// Mitsubishi GX Works2 project: Project   PLC: Q00U

PROGRAM Conveyor
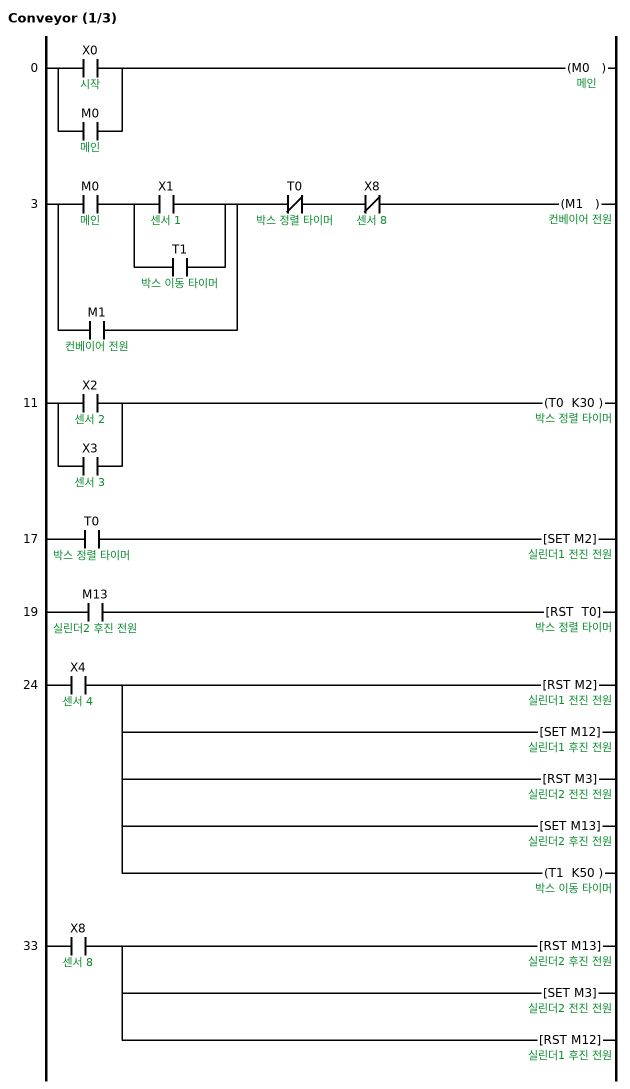
0     LD      X0  ; 시작
      OR      M0  ; 메인
      OUT     M0  ; 메인
3     LD      M0  ; 메인
      LD      X1  ; 센서 1
      OR      T1  ; 박스 이동 타이머
      ANB
      OR      M1  ; 컨베이어 전원
      ANI     T0  ; 박스 정렬 타이머
      ANI     X8  ; 센서 8
      OUT     M1  ; 컨베이어 전원
11    LD      X2  ; 센서 2
      OR      X3  ; 센서 3
      OUT     T0 K30  ; 박스 정렬 타이머
17    LD      T0  ; 박스 정렬 타이머
      SET     M2  ; 실린더1 전진 전원
19    LD      M13  ; 실린더2 후진 전원
      RST     T0  ; 박스 정렬 타이머
24    LD      X4  ; 센서 4
      RST     M2  ; 실린더1 전진 전원
      SET     M12  ; 실린더1 후진 전원
      RST     M3  ; 실린더2 전진 전원
      SET     M13  ; 실린더2 후진 전원
      OUT     T1 K50  ; 박스 이동 타이머
33    LD      X8  ; 센서 8
      RST     M13  ; 실린더2 후진 전원
      SET     M3  ; 실린더2 전진 전원
      RST     M12  ; 실린더1 후진 전원
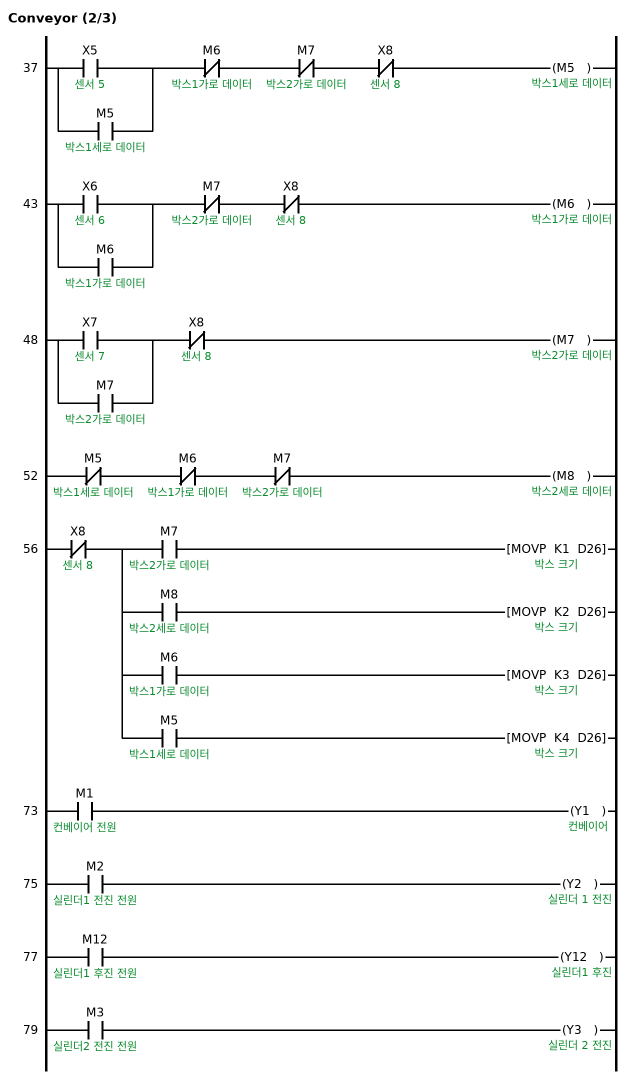
37    LD      X5  ; 센서 5
      OR      M5  ; 박스1세로 데이터
      ANI     M6  ; 박스1가로 데이터
      ANI     M7  ; 박스2가로 데이터
      ANI     X8  ; 센서 8
      OUT     M5  ; 박스1세로 데이터
43    LD      X6  ; 센서 6
      OR      M6  ; 박스1가로 데이터
      ANI     M7  ; 박스2가로 데이터
      ANI     X8  ; 센서 8
      OUT     M6  ; 박스1가로 데이터
48    LD      X7  ; 센서 7
      OR      M7  ; 박스2가로 데이터
      ANI     X8  ; 센서 8
      OUT     M7  ; 박스2가로 데이터
52    LDI     M5  ; 박스1세로 데이터
      ANI     M6  ; 박스1가로 데이터
      ANI     M7  ; 박스2가로 데이터
      OUT     M8  ; 박스2세로 데이터
56    LDI     X8  ; 센서 8
      MPS
      AND     M7  ; 박스2가로 데이터
      MOVP    K1 D26  ; 박스 크기
      MRD
      AND     M8  ; 박스2세로 데이터
      MOVP    K2 D26
      MRD
      AND     M6  ; 박스1가로 데이터
      MOVP    K3 D26
      MPP
      AND     M5  ; 박스1세로 데이터
      MOVP    K4 D26
73    LD      M1  ; 컨베이어 전원
      OUT     Y1  ; 컨베이어
75    LD      M2  ; 실린더1 전진 전원
      OUT     Y2  ; 실린더 1 전진
77    LD      M12  ; 실린더1 후진 전원
      OUT     Y12  ; 실린더1 후진
79    LD      M3  ; 실린더2 전진 전원
      OUT     Y3  ; 실린더 2 전진
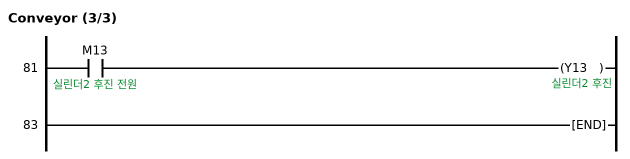
81    LD      M13  ; 실린더2 후진 전원
      OUT     Y13  ; 실린더2 후진
83    END
END_PROGRAM

PROGRAM Loading
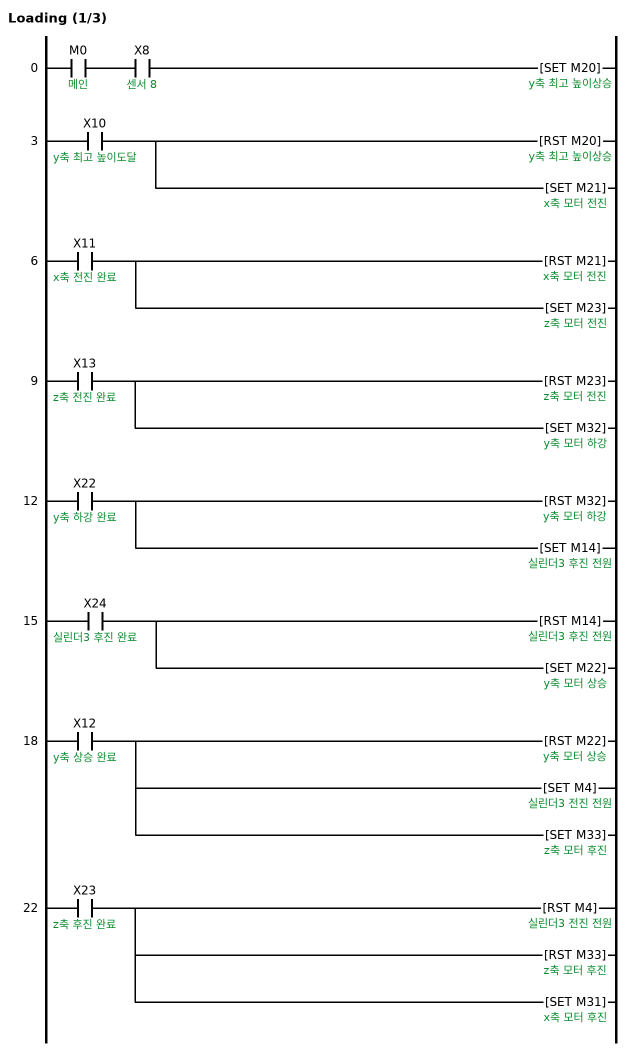
0     LD      M0  ; 메인
      AND     X8  ; 센서 8
      SET     M20  ; y축 최고 높이상승
3     LD      X10  ; y축 최고 높이도달
      RST     M20  ; y축 최고 높이상승
      SET     M21  ; x축 모터 전진
6     LD      X11  ; x축 전진 완료
      RST     M21  ; x축 모터 전진
      SET     M23  ; z축 모터 전진
9     LD      X13  ; z축 전진 완료
      RST     M23  ; z축 모터 전진
      SET     M32  ; y축 모터 하강
12    LD      X22  ; y축 하강 완료
      RST     M32  ; y축 모터 하강
      SET     M14  ; 실린더3 후진 전원
15    LD      X24  ; 실린더3 후진 완료
      RST     M14  ; 실린더3 후진 전원
      SET     M22  ; y축 모터 상승
18    LD      X12  ; y축 상승 완료
      RST     M22  ; y축 모터 상승
      SET     M4  ; 실린더3 전진 전원
      SET     M33  ; z축 모터 후진
22    LD      X23  ; z축 후진 완료
      RST     M4  ; 실린더3 전진 전원
      RST     M33  ; z축 모터 후진
      SET     M31  ; x축 모터 후진
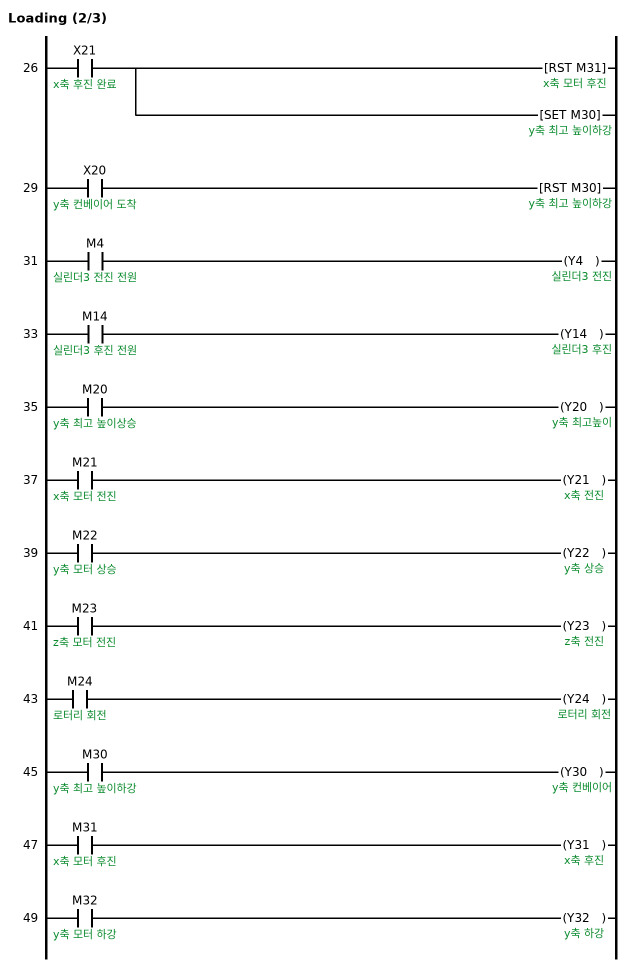
26    LD      X21  ; x축 후진 완료
      RST     M31  ; x축 모터 후진
      SET     M30  ; y축 최고 높이하강
29    LD      X20  ; y축 컨베이어 도착
      RST     M30  ; y축 최고 높이하강
31    LD      M4  ; 실린더3 전진 전원
      OUT     Y4  ; 실린더3 전진
33    LD      M14  ; 실린더3 후진 전원
      OUT     Y14  ; 실린더3 후진
35    LD      M20  ; y축 최고 높이상승
      OUT     Y20  ; y축 최고높이
37    LD      M21  ; x축 모터 전진
      OUT     Y21  ; x축 전진
39    LD      M22  ; y축 모터 상승
      OUT     Y22  ; y축 상승
41    LD      M23  ; z축 모터 전진
      OUT     Y23  ; z축 전진
43    LD      M24  ; 로터리 회전
      OUT     Y24  ; 로터리 회전
45    LD      M30  ; y축 최고 높이하강
      OUT     Y30  ; y축 컨베이어
47    LD      M31  ; x축 모터 후진
      OUT     Y31  ; x축 후진
49    LD      M32  ; y축 모터 하강
      OUT     Y32  ; y축 하강
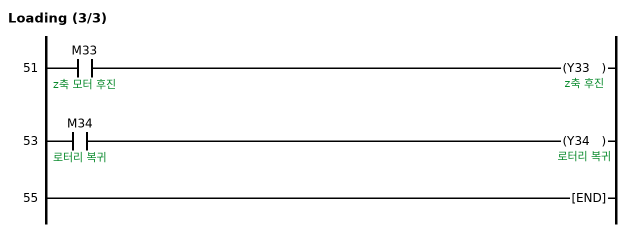
51    LD      M33  ; z축 모터 후진
      OUT     Y33  ; z축 후진
53    LD      M34  ; 로터리 복귀
      OUT     Y34  ; 로터리 복귀
55    END
END_PROGRAM

PROGRAM Step
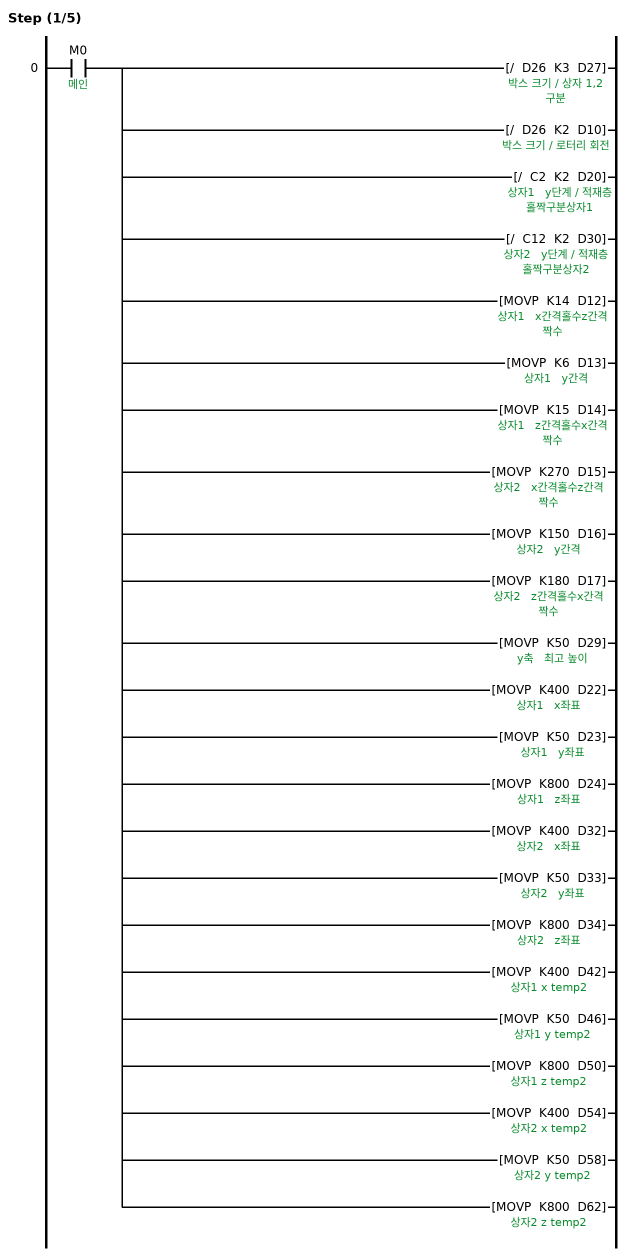
0     LD      M0  ; 메인
      /       D26 K3 D27  ; 박스 크기 / 상자 1,2 구분
      /       D26 K2 D10  ; 로터리 회전
      /       C2 K2 D20  ; 상자1   y단계 / 적재층  홀짝구분상자1
      /       C12 K2 D30  ; 상자2   y단계 / 적재층  홀짝구분상자2
      MOVP    K14 D12  ; 상자1   x간격홀수z간격짝수
      MOVP    K6 D13  ; 상자1   y간격
      MOVP    K15 D14  ; 상자1   z간격홀수x간격짝수
      MOVP    K270 D15  ; 상자2   x간격홀수z간격짝수
      MOVP    K150 D16  ; 상자2   y간격
      MOVP    K180 D17  ; 상자2   z간격홀수x간격짝수
      MOVP    K50 D29  ; y축   최고 높이
      MOVP    K400 D22  ; 상자1   x좌표
      MOVP    K50 D23  ; 상자1   y좌표
      MOVP    K800 D24  ; 상자1   z좌표
      MOVP    K400 D32  ; 상자2   x좌표
      MOVP    K50 D33  ; 상자2   y좌표
      MOVP    K800 D34  ; 상자2   z좌표
      MOVP    K400 D42  ; 상자1 x temp2
      MOVP    K50 D46  ; 상자1 y temp2
      MOVP    K800 D50  ; 상자1 z temp2
      MOVP    K400 D54  ; 상자2 x temp2
      MOVP    K50 D58  ; 상자2 y temp2
      MOVP    K800 D62  ; 상자2 z temp2
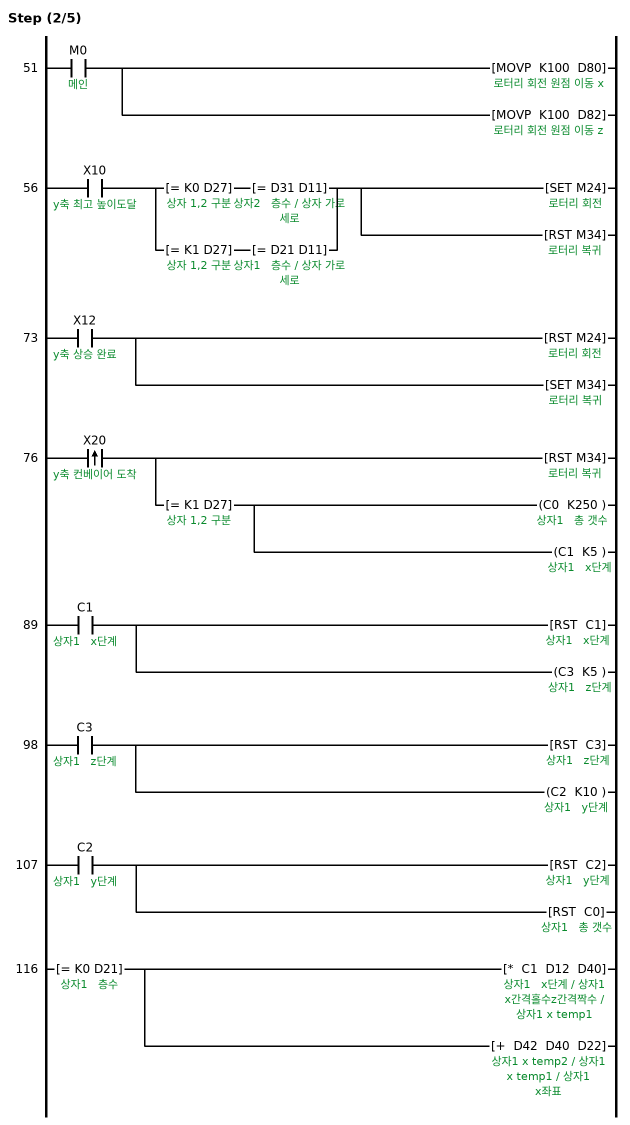
51    LD      M0  ; 메인
      MOVP    K100 D80  ; 로터리 회전 원점 이동 x
      MOVP    K100 D82  ; 로터리 회전 원점 이동 z
56    LD      X10  ; y축 최고 높이도달
      LD=     K0 D27  ; 상자 1,2 구분
      AND=    D31 D11  ; 상자2   층수 / 상자 가로 세로
      LD=     K1 D27  ; 상자 1,2 구분
      AND=    D21 D11  ; 상자1   층수 / 상자 가로 세로
      ORB
      ANB
      SET     M24  ; 로터리 회전
      RST     M34  ; 로터리 복귀
73    LD      X12  ; y축 상승 완료
      RST     M24  ; 로터리 회전
      SET     M34  ; 로터리 복귀
76    LDP     X20  ; y축 컨베이어 도착
      RST     M34  ; 로터리 복귀
      AND=    K1 D27  ; 상자 1,2 구분
      OUT     C0 K250  ; 상자1   총 갯수
      OUT     C1 K5  ; 상자1   x단계
89    LD      C1  ; 상자1   x단계
      RST     C1  ; 상자1   x단계
      OUT     C3 K5  ; 상자1   z단계
98    LD      C3  ; 상자1   z단계
      RST     C3  ; 상자1   z단계
      OUT     C2 K10  ; 상자1   y단계
107   LD      C2  ; 상자1   y단계
      RST     C2  ; 상자1   y단계
      RST     C0  ; 상자1   총 갯수
116   LD=     K0 D21  ; 상자1   층수
      *       C1 D12 D40  ; 상자1 x temp1
      +       D42 D40 D22
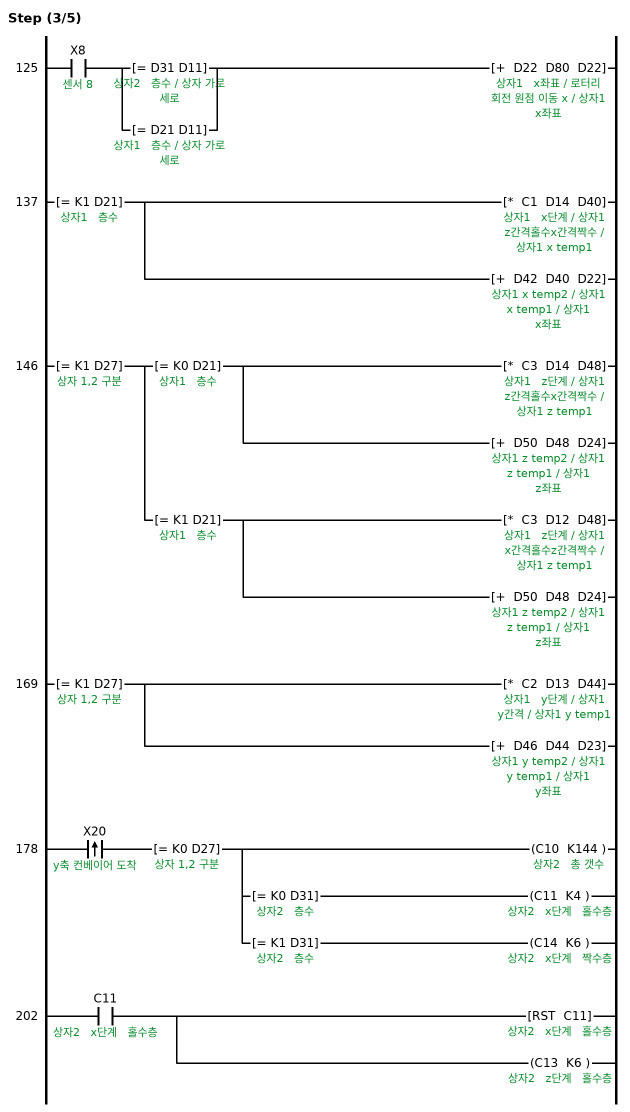
125   LD      X8  ; 센서 8
      LD=     D31 D11  ; 상자2   층수 / 상자 가로 세로
      OR=     D21 D11  ; 상자1   층수 / 상자 가로 세로
      ANB
      +       D22 D80 D22
137   LD=     K1 D21  ; 상자1   층수
      *       C1 D14 D40
      +       D42 D40 D22
146   LD=     K1 D27  ; 상자 1,2 구분
      MPS
      AND=    K0 D21  ; 상자1   층수
      *       C3 D14 D48  ; 상자1 z temp1
      +       D50 D48 D24
      MPP
      AND=    K1 D21  ; 상자1   층수
      *       C3 D12 D48
      +       D50 D48 D24
169   LD=     K1 D27  ; 상자 1,2 구분
      *       C2 D13 D44  ; 상자1 y temp1
      +       D46 D44 D23
178   LDP     X20  ; y축 컨베이어 도착
      AND=    K0 D27  ; 상자 1,2 구분
      OUT     C10 K144  ; 상자2   총 갯수
      MPS
      AND=    K0 D31  ; 상자2   층수
      OUT     C11 K4  ; 상자2   x단계   홀수층
      MPP
      AND=    K1 D31  ; 상자2   층수
      OUT     C14 K6  ; 상자2   x단계   짝수층
202   LD      C11  ; 상자2   x단계   홀수층
      RST     C11  ; 상자2   x단계   홀수층
      OUT     C13 K6  ; 상자2   z단계   홀수층
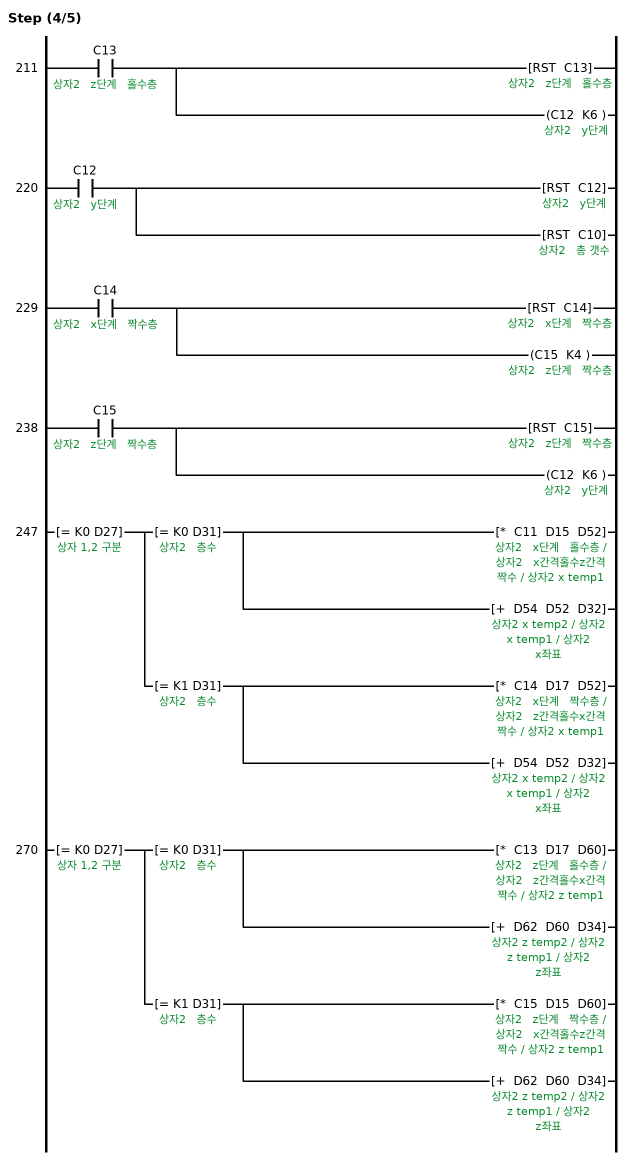
211   LD      C13  ; 상자2   z단계   홀수층
      RST     C13  ; 상자2   z단계   홀수층
      OUT     C12 K6  ; 상자2   y단계
220   LD      C12  ; 상자2   y단계
      RST     C12  ; 상자2   y단계
      RST     C10  ; 상자2   총 갯수
229   LD      C14  ; 상자2   x단계   짝수층
      RST     C14  ; 상자2   x단계   짝수층
      OUT     C15 K4  ; 상자2   z단계   짝수층
238   LD      C15  ; 상자2   z단계   짝수층
      RST     C15  ; 상자2   z단계   짝수층
      OUT     C12 K6  ; 상자2   y단계
247   LD=     K0 D27  ; 상자 1,2 구분
      MPS
      AND=    K0 D31  ; 상자2   층수
      *       C11 D15 D52  ; 상자2 x temp1
      +       D54 D52 D32
      MPP
      AND=    K1 D31  ; 상자2   층수
      *       C14 D17 D52
      +       D54 D52 D32
270   LD=     K0 D27  ; 상자 1,2 구분
      MPS
      AND=    K0 D31  ; 상자2   층수
      *       C13 D17 D60  ; 상자2 z temp1
      +       D62 D60 D34
      MPP
      AND=    K1 D31  ; 상자2   층수
      *       C15 D15 D60
      +       D62 D60 D34
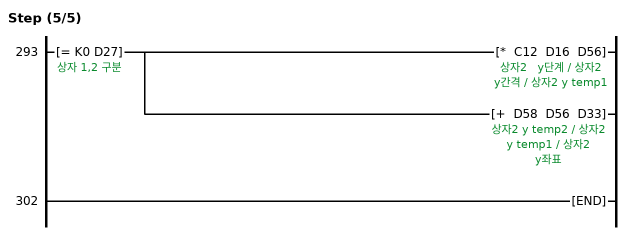
293   LD=     K0 D27  ; 상자 1,2 구분
      *       C12 D16 D56  ; 상자2 y temp1
      +       D58 D56 D33
302   END
END_PROGRAM

// device comments not shown above
X14  ; 실린더3 전진 완료
D0  ; 박스 크기
D1  ; 상자 1,2 구분
D2  ; 나머지
D3  ; 상자1 x방향 업
D4  ; 상자1 x좌표 변수
D5  ; 상자1 y방향 업
D6  ; 상자1 y좌표 변수
D7  ; 상자1 z방향 업
D8  ; 상자1 z좌표 변수
D28  ; 나머지
